ABB RAPID module: FML2H3SegmentOrg.mod

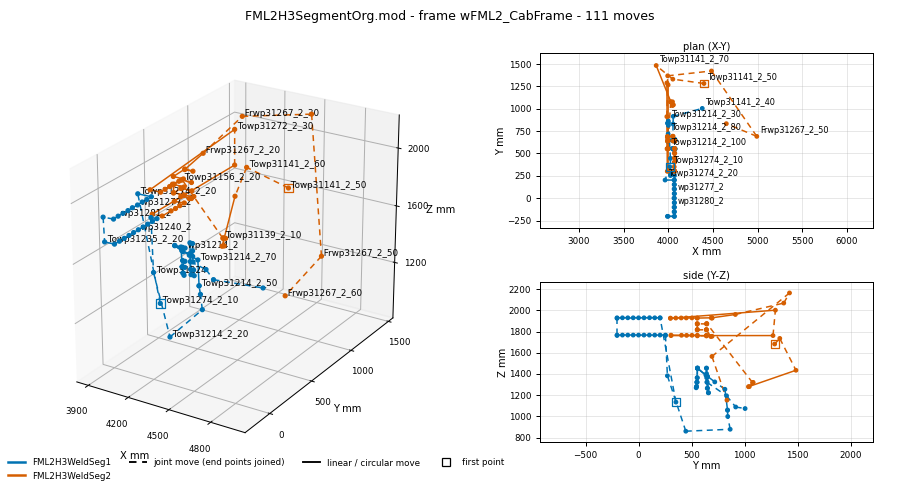
[picture p0: tool path of FML2H3SegmentOrg.mod in frame wFML2_CabFrame, 111 of 113 moves have a stored position in this frame; points joined in program order, loops and branches not executed]
%%%
   VERSION: 1
   LANGUAGE: ENGLISH
%%%

MODULE FML2H3Segment
  !
  !***********************************
  !*                                 *
  !*   Module : FML2H3Segment.mod    *
  !*   Name   : R2 2V6=V2=AR22       *
  !*   Task   : T_Rob1               *
  !*                                 *
  !***********************************
  !
  ! Rob 1 : irb 66-61388 \ 2V6=V2=AR22
  !
  !*********************
  ! Robtargets
  !*********************
  LOCAL CONST robtarget Towp31274_2_10:=[[4016.45,352.30,1134.15],[0.162794,-0.671420,0.154786,-0.706211],[0,-1,0,0],[9E9,100.000,9E9,9E9,9E9,9E9]];
  LOCAL CONST robtarget Towp31274_2_20:=[[3964.30,202.95,1926.71],[0.082443,-0.684548,0.078373,-0.720038],[-1,-1,0,0],[9E9,129.723,9E9,9E9,9E9,9E9]];
  LOCAL CONST robtarget wp31274_2:=[[4065.31,202.75,1929.60],[0.0644104,-0.686294,0.0612422,-0.721873],[-1,-1,0,0],[9E+09,25.0006,9E+09,9E+09,9E+09,9E+09]];
  LOCAL CONST robtarget Towp31275_2_10:=[[4050.21,151.97,1923.72],[0.064411,-0.686287,0.061241,-0.721867],[-1,-1,0,0],[9E9,30.000,9E9,9E9,9E9,9E9]];
  LOCAL CONST robtarget wp31275_2:=[[4065.68,152.48,1929.12],[0.0643992,-0.686292,0.0612485,-0.721875],[-1,-1,0,0],[9E+09,25.0001,9E+09,9E+09,9E+09,9E+09]];
  LOCAL CONST robtarget Towp31276_2_10:=[[4050.21,101.31,1923.72],[0.090401,-0.683647,0.085941,-0.719087],[-1,-1,0,0],[9E9,30.000,9E9,9E9,9E9,9E9]];
  LOCAL CONST robtarget wp31276_2:=[[4065.38,103.38,1930.02],[0.105651,-0.68166,0.100447,-0.716999],[-1,-1,0,0],[9E+09,25.001,9E+09,9E+09,9E+09,9E+09]];
  LOCAL CONST robtarget Towp31277_2_10:=[[4050.21,50.65,1923.72],[0.105651,-0.681667,0.100451,-0.717007],[-1,-1,0,0],[9E9,30.000,9E9,9E9,9E9,9E9]];
  LOCAL CONST robtarget wp31277_2:=[[4066.10,51.42,1929.09],[0.105652,-0.681659,0.100451,-0.717],[-1,-1,0,0],[9E+09,24.9997,9E+09,9E+09,9E+09,9E+09]];
  LOCAL CONST robtarget Towp31278_2_10:=[[4050.21,0.00,1923.72],[0.115181,-0.680257,0.109501,-0.715537],[-1,-1,0,0],[9E9,30.000,9E9,9E9,9E9,9E9]];
  LOCAL CONST robtarget wp31278_2:=[[4063.93,-0.02,1929.13],[0.115181,-0.680257,0.109501,-0.715537],[-1,-1,0,0],[9E9,25.000,9E9,9E9,9E9,9E9]];
  LOCAL CONST robtarget Towp31279_2_10:=[[4050.21,-50.65,1923.72],[0.131391,-0.677597,0.124921,-0.712737],[-1,-1,0,0],[9E9,30.000,9E9,9E9,9E9,9E9]];
  LOCAL CONST robtarget wp31279_2:=[[4066.40,-50.84,1929.14],[0.131392,-0.677596,0.124922,-0.712737],[-1,-1,0,0],[9E+09,25.0001,9E+09,9E+09,9E+09,9E+09]];
  LOCAL CONST robtarget Towp31280_2_10:=[[4050.21,-101.31,1923.72],[0.131391,-0.677597,0.124921,-0.712737],[-1,-1,0,0],[9E9,30.000,9E9,9E9,9E9,9E9]];
  LOCAL CONST robtarget wp31280_2:=[[4064.89,-101.49,1929.14],[0.131386,-0.677595,0.124923,-0.712739],[-1,-1,0,0],[9E+09,25.0001,9E+09,9E+09,9E+09,9E+09]];
  LOCAL CONST robtarget Towp31281_2_10:=[[4050.21,-151.97,1923.72],[0.144731,-0.675137,0.137601,-0.710147],[-1,-1,0,0],[9E9,30.000,9E9,9E9,9E9,9E9]];
  LOCAL CONST robtarget wp31281_2:=[[4065.09,-152.28,1929.13],[0.144727,-0.675136,0.137603,-0.710148],[-1,-1,0,0],[9E+09,25.0001,9E+09,9E+09,9E+09,9E+09]];
  LOCAL CONST robtarget Towp31282_2_10:=[[4050.21,-202.63,1923.72],[0.172142,-0.669297,0.163652,-0.704007],[-1,-1,0,0],[9E9,30.000,9E9,9E9,9E9,9E9]];
  LOCAL CONST robtarget wp31282_2:=[[4067.03,-203.17,1929.08],[0.16373,-0.671199,0.155666,-0.706012],[-1,-1,0,0],[9E+09,25.0001,9E+09,9E+09,9E+09,9E+09]];
  LOCAL CONST robtarget Towp31235_2_10:=[[3990.48,-202.94,1924.40],[0.146426,-0.674805,0.139211,-0.709801],[-1,-1,0,0],[9E9,100.000,9E9,9E9,9E9,9E9]];
  LOCAL CONST robtarget Towp31235_2_20:=[[3996.84,-202.94,1763.15],[0.141411,-0.692597,0.141321,-0.693067],[-1,-1,0,0],[9E9,100.000,9E9,9E9,9E9,9E9]];
  LOCAL CONST robtarget wp31235_2:=[[4069.18,-202.99,1765.78],[0.141408,-0.692595,0.141328,-0.693067],[-1,-1,0,0],[9E+09,25.0001,9E+09,9E+09,9E+09,9E+09]];
  LOCAL CONST robtarget Towp31236_2_10:=[[4054.42,-151.97,1759.49],[0.128101,-0.695197,0.128011,-0.695637],[-1,-1,0,0],[9E9,30.000,9E9,9E9,9E9,9E9]];
  LOCAL CONST robtarget wp31236_2:=[[4069.77,-152.16,1766.20],[0.128108,-0.695197,0.128004,-0.695632],[-1,-1,0,0],[9E+09,25.0001,9E+09,9E+09,9E+09,9E+09]];
  LOCAL CONST robtarget Towp31237_2_10:=[[4054.42,-101.31,1759.49],[0.128101,-0.695197,0.128011,-0.695637],[-1,-1,0,0],[9E9,30.000,9E9,9E9,9E9,9E9]];
  LOCAL CONST robtarget wp31237_2:=[[4070.38,-101.50,1766.20],[0.1281,-0.695194,0.128011,-0.695635],[-1,-1,0,0],[9E+09,24.9996,9E+09,9E+09,9E+09,9E+09]];
  LOCAL CONST robtarget Towp31238_2_10:=[[4054.41,-50.65,1759.49],[0.128381,-0.695127,0.128301,-0.695597],[-1,-1,0,0],[9E9,30.000,9E9,9E9,9E9,9E9]];
  LOCAL CONST robtarget wp31238_2:=[[4070.05,-50.84,1766.20],[0.128385,-0.695128,0.128301,-0.695595],[-1,-1,0,0],[9E+09,24.9986,9E+09,9E+09,9E+09,9E+09]];
  LOCAL CONST robtarget Towp31239_2_10:=[[4054.41,0.00,1759.49],[0.128101,-0.695197,0.128011,-0.695637],[-1,-1,0,0],[9E9,30.000,9E9,9E9,9E9,9E9]];
  LOCAL CONST robtarget wp31239_2:=[[4069.17,-0.19,1766.20],[0.128107,-0.695196,0.128006,-0.695633],[-1,-1,0,0],[9E+09,25.0001,9E+09,9E+09,9E+09,9E+09]];
  LOCAL CONST robtarget Towp31240_2_10:=[[4054.42,50.65,1759.49],[0.113601,-0.697707,0.113531,-0.698147],[-1,-1,0,0],[9E9,30.000,9E9,9E9,9E9,9E9]];
  LOCAL CONST robtarget wp31240_2:=[[4069.38,50.63,1766.22],[0.113599,-0.697707,0.113531,-0.698148],[-1,-1,0,0],[9E+09,24.9996,9E+09,9E+09,9E+09,9E+09]];
  LOCAL CONST robtarget Towp31241_2_10:=[[4054.42,101.31,1759.49],[0.113601,-0.697707,0.113531,-0.698147],[-1,-1,0,0],[9E9,30.000,9E9,9E9,9E9,9E9]];
  LOCAL CONST robtarget wp31241_2:=[[4070.30,101.27,1766.21],[0.113606,-0.697708,0.113529,-0.698146],[-1,-1,0,0],[9E+09,25.0001,9E+09,9E+09,9E+09,9E+09]];
  LOCAL CONST robtarget Towp31242_2_10:=[[4054.42,151.97,1759.49],[0.062941,-0.704077,0.062901,-0.704527],[-1,-1,0,0],[9E9,30.000,9E9,9E9,9E9,9E9]];
  LOCAL CONST robtarget wp31242_2:=[[4069.10,152.47,1766.17],[0.0629363,-0.704074,0.0629048,-0.704529],[-1,-1,0,0],[9E+09,25.0006,9E+09,9E+09,9E+09,9E+09]];
  LOCAL CONST robtarget Towp31243_2_10:=[[4054.42,202.62,1759.49],[0.113601,-0.697707,0.113531,-0.698147],[-1,-1,0,0],[9E9,30.000,9E9,9E9,9E9,9E9]];
  LOCAL CONST robtarget wp31243_2:=[[4069.64,202.57,1766.21],[0.113604,-0.697709,0.113531,-0.698146],[-1,-1,0,0],[9E+09,25.0006,9E+09,9E+09,9E+09,9E+09]];
  LOCAL CONST robtarget Towp31244_2_10:=[[4054.42,253.28,1759.49],[0.098771,-0.699977,0.098711,-0.700377],[-1,-1,0,0],[9E9,30.000,9E9,9E9,9E9,9E9]];
  LOCAL CONST robtarget wp31244_2:=[[4069.47,253.41,1766.22],[0.098779,-0.699981,0.0987012,-0.700377],[-1,-1,0,0],[9E+09,25.0001,9E+09,9E+09,9E+09,9E+09]];
  LOCAL CONST robtarget Towp31214_2_10:=[[4024.34,253.56,1763.19],[0.085541,-0.701915,0.085526,-0.701914],[-1,-1,0,0],[9E9,100.000,9E9,9E9,9E9,9E9]];
  LOCAL CONST robtarget Towp31214_2_20:=[[4024.15,445.26,859.90],[0.209663,-0.669229,0.163293,-0.693909],[0,-1,0,0],[9E9,30.000,9E9,9E9,9E9,9E9]];
  LOCAL CONST robtarget Towp31214_2_30:=[[4000.53,863.67,878.09],[0.209664,-0.669228,0.163288,-0.693910],[0,-1,1,0],[9E9,29.999,9E9,9E9,9E9,9E9]];
  LOCAL CONST robtarget Towp31214_2_40:=[[4001.68,840.75,998.57],[0.206529,-0.679094,0.209107,-0.672645],[0,-1,0,0],[9E9,74.423,9E9,9E9,9E9,9E9]];
  LOCAL CONST robtarget Towp31214_2_50:=[[3992.94,838.76,1058.72],[0.202837,-0.683610,0.236031,-0.660170],[0,-1,0,0],[9E9,99.999,9E9,9E9,9E9,9E9]];
  LOCAL CONST robtarget Towp31214_2_60:=[[3992.93,838.76,1058.72],[0.202842,-0.683617,0.236032,-0.660177],[0,-1,0,0],[9E9,100.000,9E9,9E9,9E9,9E9]];
  LOCAL CONST robtarget Towp31214_2_70:=[[4001.18,814.12,1255.53],[0.202842,-0.683617,0.236032,-0.660147],[0,-1,0,0],[9E9,100.000,9E9,9E9,9E9,9E9]];
  LOCAL CONST robtarget Towp31214_2_80:=[[3998.59,718.55,1324.71],[0.238582,-0.667717,0.261043,-0.655047],[-1,-1,0,0],[9E9,100.000,9E9,9E9,9E9,9E9]];
  LOCAL CONST robtarget Towp31214_2_90:=[[3996.43,634.65,1388.99],[0.301443,-0.639626,0.301443,-0.639626],[-1,0,-1,0],[9E9,100.000,9E9,9E9,9E9,9E9]];
  LOCAL CONST robtarget Towp31214_2_100:=[[3996.43,555.21,1454.56],[0.301443,-0.639626,0.301443,-0.639626],[-1,0,-1,0],[9E9,100.000,9E9,9E9,9E9,9E9]];
  LOCAL CONST robtarget wp31214_2:=[[4074.78,555.19,1454.58],[0.301448,-0.639635,0.301446,-0.63963],[-1,-1,0,0],[9E+09,25.0006,9E+09,9E+09,9E+09,9E+09]];
  LOCAL CONST robtarget Towp31216_2_10:=[[4055.43,555.21,1454.56],[0.301443,-0.639626,0.301443,-0.639626],[-1,0,-1,0],[9E9,30.000,9E9,9E9,9E9,9E9]];
  LOCAL CONST robtarget Towp31216_2_20:=[[4055.43,553.86,1363.93],[0.301443,-0.639626,0.301443,-0.639626],[-1,-1,0,0],[9E9,30.000,9E9,9E9,9E9,9E9]];
  LOCAL CONST robtarget wp31216_2:=[[4074.88,551.89,1363.92],[0.30144,-0.639615,0.301463,-0.639645],[-1,-1,0,0],[9E+09,25.0011,9E+09,9E+09,9E+09,9E+09]];
  LOCAL CONST robtarget Towp31217_2_10:=[[4053.93,550.53,1320.87],[0.301443,-0.639626,0.301443,-0.639626],[-1,-1,0,0],[9E9,30.000,9E9,9E9,9E9,9E9]];
  LOCAL CONST robtarget wp31217_2:=[[4074.70,550.51,1322.31],[0.301448,-0.639642,0.301439,-0.639626],[-1,-1,0,0],[9E+09,25.0006,9E+09,9E+09,9E+09,9E+09]];
  LOCAL CONST robtarget Towp31218_2_10:=[[4053.93,550.53,1320.87],[0.301443,-0.639626,0.301443,-0.639626],[-1,-1,0,0],[9E9,30.000,9E9,9E9,9E9,9E9]];
  LOCAL CONST robtarget Towp31218_2_20:=[[4066.88,546.50,1280.56],[0.414899,-0.572588,0.414893,-0.572595],[-1,0,-1,0],[9E9,29.999,9E9,9E9,9E9,9E9]];
  LOCAL CONST robtarget wp31218_2:=[[4072.69,543.03,1269.14],[0.414899,-0.572585,0.414894,-0.572598],[-1,0,-1,0],[9E+09,24.9991,9E+09,9E+09,9E+09,9E+09]];
  LOCAL CONST robtarget Towp31143_2_10:=[[4060.85,546.50,1280.50],[0.414897,-0.572601,0.414893,-0.572583],[-1,0,-1,0],[9E9,30.000,9E9,9E9,9E9,9E9]];
  LOCAL CONST robtarget Towp31143_2_20:=[[4043.07,555.22,1454.48],[0.301450,-0.639637,0.301445,-0.639627],[-1,-1,0,0],[9E9,56.519,9E9,9E9,9E9,9E9]];
  LOCAL CONST robtarget Towp31143_2_30:=[[3996.29,555.12,1452.38],[0.302913,-0.638946,0.302913,-0.638946],[-1,0,-1,0],[9E9,100.000,9E9,9E9,9E9,9E9]];
  LOCAL CONST robtarget Towp31143_2_40:=[[3996.29,649.96,1374.83],[0.302913,-0.638946,0.302913,-0.638946],[-1,0,-1,0],[9E9,100.000,9E9,9E9,9E9,9E9]];
  LOCAL CONST robtarget Towp31143_2_50:=[[4049.79,649.96,1374.83],[0.302913,-0.638946,0.302913,-0.638946],[-1,0,-1,0],[9E9,100.000,9E9,9E9,9E9,9E9]];
  LOCAL CONST robtarget Towp31143_2_60:=[[4048.93,659.76,1222.18],[0.404844,-0.579746,0.404844,-0.579746],[-1,0,-1,0],[9E9,30.000,9E9,9E9,9E9,9E9]];
  LOCAL CONST robtarget wp31143_2:=[[4074.64,657.65,1222.13],[0.404851,-0.579739,0.404851,-0.579737],[-1,0,-1,0],[9E+09,25.0006,9E+09,9E+09,9E+09,9E+09]];
  LOCAL CONST robtarget Towp31144_2_10:=[[4055.00,650.35,1263.04],[0.404844,-0.579746,0.404844,-0.579746],[-1,0,-1,0],[9E9,30.000,9E9,9E9,9E9,9E9]];
  LOCAL CONST robtarget wp31144_2:=[[4075.34,650.28,1265.40],[0.404844,-0.579734,0.40484,-0.579754],[-1,0,-1,0],[9E+09,25.0006,9E+09,9E+09,9E+09,9E+09]];
  LOCAL CONST robtarget Towp31148_2_10:=[[4053.93,647.44,1265.33],[0.404844,-0.579746,0.404844,-0.579746],[-1,0,-1,0],[9E9,30.000,9E9,9E9,9E9,9E9]];
  LOCAL CONST robtarget Towp31148_2_20:=[[4055.43,640.80,1454.56],[0.301443,-0.639626,0.301443,-0.639626],[-1,0,-1,0],[9E9,30.000,9E9,9E9,9E9,9E9]];
  LOCAL CONST robtarget wp31148_2:=[[4075.85,639.45,1454.59],[0.30144,-0.639621,0.301448,-0.639647],[-1,0,-1,0],[9E+09,24.9996,9E+09,9E+09,9E+09,9E+09]];
  LOCAL CONST robtarget Towp31147_2_10:=[[4056.50,644.08,1399.66],[0.301443,-0.639626,0.301443,-0.639626],[-1,0,-1,0],[9E9,30.000,9E9,9E9,9E9,9E9]];
  LOCAL CONST robtarget wp31147_2:=[[4075.11,640.62,1402.76],[0.301453,-0.639626,0.301456,-0.639632],[-1,-1,0,0],[9E+09,25.0011,9E+09,9E+09,9E+09,9E+09]];
  LOCAL CONST robtarget Towp31146_2_10:=[[4056.50,644.14,1360.80],[0.301443,-0.639626,0.301443,-0.639626],[-1,0,-1,0],[9E9,30.000,9E9,9E9,9E9,9E9]];
  LOCAL CONST robtarget wp31146_2:=[[4074.31,642.12,1363.96],[0.301442,-0.639624,0.30145,-0.639641],[-1,-1,0,0],[9E+09,25.0006,9E+09,9E+09,9E+09,9E+09]];
  LOCAL CONST robtarget Towp31145_2_10:=[[4055.00,647.57,1317.86],[0.329033,-0.625896,0.329033,-0.625896],[-1,0,-1,0],[9E9,30.000,9E9,9E9,9E9,9E9]];
  LOCAL CONST robtarget wp31145_2:=[[4075.02,645.18,1323.40],[0.329045,-0.625872,0.329049,-0.625892],[-1,0,-1,0],[9E+09,25.0001,9E+09,9E+09,9E+09,9E+09]];
  LOCAL CONST robtarget Towp31141_2_10:=[[4053.93,645.31,1320.69],[0.329033,-0.625896,0.329033,-0.625896],[-1,0,-1,0],[9E9,30.000,9E9,9E9,9E9,9E9]];
  LOCAL CONST robtarget Towp31141_2_20:=[[4053.93,829.43,1193.98],[0.329033,-0.625896,0.329033,-0.625896],[-1,0,-1,0],[9E9,50.000,9E9,9E9,9E9,9E9]];
  LOCAL CONST robtarget Towp31141_2_30:=[[4055.61,915.71,1088.15],[0.311158,-0.574108,0.357827,-0.667488],[-1,0,-1,0],[9E9,49.997,9E9,9E9,9E9,9E9]];
  LOCAL CONST robtarget Towp31141_2_40:=[[4380.43,1004.47,1073.50],[0.329033,-0.625896,0.329033,-0.625896],[-1,0,-1,0],[9E9,50.000,9E9,9E9,9E9,9E9]];
  LOCAL CONST robtarget Towp31141_2_50:=[[4399.60,1283.05,1681.87],[0.242317,-0.631638,0.388427,-0.625652],[-2,0,-1,0],[9E9,48.091,9E9,9E9,9E9,9E9]];
  LOCAL CONST robtarget Towp31141_2_60:=[[4051.14,1331.48,1734.78],[0.322441,-0.595529,0.421583,-0.603029],[-2,0,-1,0],[9E9,48.372,9E9,9E9,9E9,9E9]];
  LOCAL CONST robtarget Towp31141_2_70:=[[3865.02,1484.04,1434.51],[0.607774,-0.566534,0.442110,-0.337919],[-2,0,-2,0],[9E9,66.407,9E9,9E9,9E9,9E9]];
  LOCAL CONST robtarget Towp31141_2_80:=[[4046.26,1036.05,1279.43],[0.624891,-0.566993,0.438571,-0.309331],[-2,0,-2,0],[9E9,105.850,9E9,9E9,9E9,9E9]];
  LOCAL CONST robtarget wp31141_2:=[[4057.63,1044.03,1280.67],[0.624912,-0.586047,0.421153,-0.297766],[-2,0,-2,0],[9E+09,25.0006,9E+09,9E+09,9E+09,9E+09]];
  LOCAL CONST robtarget Towp31139_2_10:=[[4028.65,1078.45,1319.83],[0.493609,-0.505141,0.494963,-0.506156],[-2,0,-2,0],[9E+09,40,9E+09,9E+09,9E+09,9E+09]];
  LOCAL CONST robtarget wp31139_2:=[[4047.28,1078.46,1319.97],[0.493612,-0.505140,0.494959,-0.506158],[-2,0,-2,0],[9E9,25.000,9E9,9E9,9E9,9E9]];
  LOCAL CONST robtarget Towp31156_2_10:=[[4027.10,1076.22,1316.29],[0.496076,-0.505810,0.494748,-0.503278],[-2,0,-2,0],[9E9,82.552,9E9,9E9,9E9,9E9]];
  LOCAL CONST robtarget Towp31156_2_20:=[[3999.20,643.27,1874.83],[0.41306,-0.570139,0.400218,-0.586642],[-1,0,-1,0],[9E+09,128.149,9E+09,9E+09,9E+09,9E+09]];
  LOCAL CONST robtarget wp31156_2:=[[4071.98,640.13,1872.87],[0.413058,-0.570143,0.400228,-0.586633],[-1,0,-1,0],[9E+09,24.998,9E+09,9E+09,9E+09,9E+09]];
  LOCAL CONST robtarget Towp31206_2_10:=[[3993.72,643.17,1870.74],[0.413056,-0.570144,0.40022,-0.586639],[-1,0,-1,0],[9E+09,100.002,9E+09,9E+09,9E+09,9E+09]];
  LOCAL CONST robtarget Towp31206_2_20:=[[3986.60,552.91,1873.31],[0.420259,-0.563937,0.407544,-0.582465],[-1,0,-1,0],[9E+09,100.001,9E+09,9E+09,9E+09,9E+09]];
  LOCAL CONST robtarget wp31206_2:=[[4072.95,553.58,1873.34],[0.420258,-0.563936,0.40753,-0.582476],[-1,0,-1,0],[9E+09,25.1416,9E+09,9E+09,9E+09,9E+09]];
  LOCAL CONST robtarget Towp31207_2_10:=[[3992.65,553.82,1869.80],[0.420261,-0.563933,0.407546,-0.582466],[-1,0,-1,0],[9E9,100.000,9E9,9E9,9E9,9E9]];
  LOCAL CONST robtarget Towp31207_2_20:=[[3993.78,553.55,1816.78],[0.448931,-0.544821,0.443606,-0.552127],[-1,0,-1,0],[9E+09,100.001,9E+09,9E+09,9E+09,9E+09]];
  LOCAL CONST robtarget wp31207_2:=[[4071.90,554.05,1818.23],[0.448933,-0.544814,0.443612,-0.552128],[-1,0,-1,0],[9E+09,25.0015,9E+09,9E+09,9E+09,9E+09]];
  LOCAL CONST robtarget Towp31155_2_10:=[[3993.78,552.83,1815.08],[0.448933,-0.544818,0.443605,-0.55213],[-1,0,-1,0],[9E+09,99.9996,9E+09,9E+09,9E+09,9E+09]];
  LOCAL CONST robtarget Towp31155_2_20:=[[3993.77,638.71,1816.62],[0.431159,-0.559379,0.425412,-0.56588],[-1,0,-1,0],[9E+09,100.001,9E+09,9E+09,9E+09,9E+09]];
  LOCAL CONST robtarget wp31155_2:=[[4074.77,639.89,1817.01],[0.431155,-0.559381,0.425402,-0.56589],[-1,0,-1,0],[9E+09,24.9996,9E+09,9E+09,9E+09,9E+09]];
  LOCAL CONST robtarget Towp31250_2_10:=[[3993.76,638.70,1816.62],[0.431161,-0.559377,0.425412,-0.565881],[-1,0,-1,0],[9E+09,100.001,9E+09,9E+09,9E+09,9E+09]];
  LOCAL CONST robtarget Towp31250_2_20:=[[3989.70,680.85,1752.63],[0.515328,-0.560652,0.415979,-0.497059],[-2,0,-2,0],[9E9,100.000,9E9,9E9,9E9,9E9]];
  LOCAL CONST robtarget wp31250_2:=[[4054.17,692.94,1754.95],[0.499526,-0.571079,0.416555,-0.500823],[-2,0,-2,0],[9E+09,4.63808,9E+09,9E+09,9E+09,9E+09]];
  LOCAL CONST robtarget Towp31154_10:=[[4054.88,639.53,1759.33],[0.449086,-0.544740,0.445578,-0.550491],[-1,0,-1,0],[9E9,30.000,9E9,9E9,9E9,9E9]];
  LOCAL CONST robtarget wp31154:=[[4071.23,639.50,1763.81],[0.446935,-0.546472,0.443467,-0.552227],[-1,0,-1,0],[9E+09,25.0011,9E+09,9E+09,9E+09,9E+09]];
  LOCAL CONST robtarget Towp31208_2_10:=[[3990.99,639.69,1758.85],[0.440179,-0.551840,0.436783,-0.557616],[-1,0,-1,0],[9E9,100.000,9E9,9E9,9E9,9E9]];
  LOCAL CONST robtarget Towp31208_2_20:=[[3998.00,554.01,1758.87],[0.436139,-0.555460,0.431739,-0.561113],[-1,0,-1,0],[9E9,100.000,9E9,9E9,9E9,9E9]];
  LOCAL CONST robtarget wp31208_2:=[[4073.29,554.09,1764.50],[0.418898,-0.568302,0.414662,-0.574119],[-1,0,-1,0],[9E+09,24.9991,9E+09,9E+09,9E+09,9E+09]];
  LOCAL CONST robtarget Towp31249_2_10:=[[4054.40,506.52,1759.39],[0.420905,-0.568114,0.420622,-0.568473],[-1,0,-1,0],[9E9,30.000,9E9,9E9,9E9,9E9]];
  LOCAL CONST robtarget wp31249_2:=[[4073.14,503.35,1764.12],[0.445274,-0.549243,0.444983,-0.549594],[-1,0,-1,0],[9E+09,25.0011,9E+09,9E+09,9E+09,9E+09]];
  LOCAL CONST robtarget Towp31248_2_10:=[[4054.35,455.87,1759.37],[0.442975,-0.551095,0.442670,-0.551462],[-1,0,-1,0],[9E9,30.000,9E9,9E9,9E9,9E9]];
  LOCAL CONST robtarget wp31248_2:=[[4074.33,452.68,1763.43],[0.443095,-0.550993,0.4428,-0.551364],[-1,0,-1,0],[9E+09,25.0006,9E+09,9E+09,9E+09,9E+09]];
  LOCAL CONST robtarget Towp31247_2_10:=[[4054.43,405.23,1759.44],[0.433900,-0.558272,0.433608,-0.558612],[-1,0,-1,0],[9E9,30.000,9E9,9E9,9E9,9E9]];
  LOCAL CONST robtarget wp31247_2:=[[4072.88,404.67,1764.30],[0.44457,-0.549815,0.444266,-0.550171],[-1,0,-1,0],[9E+09,25.0006,9E+09,9E+09,9E+09,9E+09]];
  LOCAL CONST robtarget Towp31245_2_10:=[[4054.33,308.91,1759.42],[0.445533,-0.549029,0.445229,-0.549398],[-1,0,-1,0],[9E9,30.000,9E9,9E9,9E9,9E9]];
  LOCAL CONST robtarget wp31245_2:=[[4073.04,305.67,1765.58],[0.442311,-0.551633,0.442006,-0.55199],[-1,0,-1,0],[9E+09,25.0011,9E+09,9E+09,9E+09,9E+09]];
  LOCAL CONST robtarget Towp31272_2_10:=[[3998.39,305.75,1761.34],[0.443862,-0.550393,0.443569,-0.550727],[-1,0,-1,0],[9E9,100.000,9E9,9E9,9E9,9E9]];
  LOCAL CONST robtarget Towp31272_2_20:=[[3998.33,1267.50,1761.67],[0.408729,-0.576926,0.408449,-0.577292],[-2,0,-2,0],[9E9,100.000,9E9,9E9,9E9,9E9]];
  LOCAL CONST robtarget Towp31272_2_30:=[[3984.69,1290.11,2001.11],[0.485005,-0.510893,0.428801,-0.565586],[-2,0,-2,0],[9E9,99.999,9E9,9E9,9E9,9E9]];
  LOCAL CONST robtarget Towp31272_2_40:=[[3989.09,300.38,1924.69],[0.521335,-0.478625,0.495645,-0.503455],[-1,0,-1,0],[9E9,100.000,9E9,9E9,9E9,9E9]];
  LOCAL CONST robtarget wp31272_2:=[[4067.79,300.37,1925.97],[0.521332,-0.478634,0.495635,-0.503456],[-1,0,-1,0],[9E+09,25.0001,9E+09,9E+09,9E+09,9E+09]];
  LOCAL CONST robtarget Towp31271_2_10:=[[4050.21,354.61,1923.72],[0.521335,-0.478645,0.495645,-0.503455],[-1,0,-1,0],[9E9,30.000,9E9,9E9,9E9,9E9]];
  LOCAL CONST robtarget wp31271_2:=[[4066.84,351.01,1926.91],[0.521334,-0.478636,0.495637,-0.503451],[-1,0,-1,0],[9E+09,25.0001,9E+09,9E+09,9E+09,9E+09]];
  LOCAL CONST robtarget Towp31270_2_10:=[[4050.21,405.27,1923.72],[0.521335,-0.478645,0.495645,-0.503455],[-1,0,-1,0],[9E9,30.000,9E9,9E9,9E9,9E9]];
  LOCAL CONST robtarget wp31270_2:=[[4066.97,401.71,1927.73],[0.521328,-0.478638,0.495633,-0.503458],[-1,0,-1,0],[9E+09,25.0001,9E+09,9E+09,9E+09,9E+09]];
  LOCAL CONST robtarget Towp31269_2_10:=[[4050.21,455.93,1923.72],[0.521335,-0.478645,0.495645,-0.503455],[-1,0,-1,0],[9E9,30.000,9E9,9E9,9E9,9E9]];
  LOCAL CONST robtarget wp31269_2:=[[4068.97,449.38,1927.88],[0.521329,-0.478638,0.495635,-0.503456],[-1,0,-1,0],[9E+09,25.0001,9E+09,9E+09,9E+09,9E+09]];
  LOCAL CONST robtarget Towp31268_2_10:=[[4050.21,506.59,1923.72],[0.521335,-0.478645,0.495645,-0.503455],[-1,0,-1,0],[9E9,30.000,9E9,9E9,9E9,9E9]];
  LOCAL CONST robtarget wp31268_2:=[[4068.26,502.99,1928.11],[0.521335,-0.478633,0.495632,-0.503457],[-1,0,-1,0],[9E+09,25.0006,9E+09,9E+09,9E+09,9E+09]];
  LOCAL CONST robtarget Towp31205_2_10:=[[4051.57,557.20,1924.47],[0.517945,-0.481745,0.487075,-0.512265],[-1,0,-1,0],[9E9,30.000,9E9,9E9,9E9,9E9]];
  LOCAL CONST robtarget wp31205_2:=[[4069.45,552.93,1926.78],[0.517952,-0.48173,0.487074,-0.51227],[-1,0,-1,0],[9E+09,25.0011,9E+09,9E+09,9E+09,9E+09]];
  LOCAL CONST robtarget Towp31267_2_10:=[[3993.41,553.66,1926.43],[0.517945,-0.481745,0.487075,-0.512265],[-1,0,-1,0],[9E9,100.000,9E9,9E9,9E9,9E9]];
  LOCAL CONST robtarget Towp31267_2_20:=[[3990.15,691.03,1929.16],[0.571776,-0.495345,0.491885,-0.430994],[-2,0,-2,0],[9E9,100.000,9E9,9E9,9E9,9E9]];
  LOCAL CONST robtarget wp31267_2:=[[4048.88,693.20,1926.26],[0.571776,-0.495344,0.491883,-0.430997],[-2,0,-2,0],[9E9,24.999,9E9,9E9,9E9,9E9]];
  LOCAL CONST robtarget Frwp31267_2_10:=[[3992.59,685.11,1928.11],[0.571776,-0.495345,0.491885,-0.430994],[-2,0,-2,0],[9E9,100.000,9E9,9E9,9E9,9E9]];
  LOCAL CONST robtarget Frwp31267_2_20:=[[3984.19,912.55,1960.54],[0.515098,-0.552535,0.426442,-0.497521],[-2,0,-2,0],[9E9,100.001,9E9,9E9,9E9,9E9]];
  LOCAL CONST robtarget Frwp31267_2_30:=[[3993.68,1368.95,2068.12],[0.440251,-0.613027,0.356615,-0.550638],[-2,0,-2,0],[9E9,100.000,9E9,9E9,9E9,9E9]];
  LOCAL CONST robtarget Frwp31267_2_40:=[[4483.73,1423.17,2163.62],[0.282020,-0.710709,0.244498,-0.596303],[-2,0,-1,0],[9E9,99.999,9E9,9E9,9E9,9E9]];
  LOCAL CONST robtarget Frwp31267_2_50:=[[4990.52,691.63,1564.75],[0.303425,-0.707680,0.184932,-0.610674],[-1,-1,0,0],[9E9,29.997,9E9,9E9,9E9,9E9]];
  LOCAL CONST robtarget Frwp31267_2_60:=[[4649.39,833.49,1152.96],[0.385471,-0.603349,-0.013916,-0.697989],[0,-1,0,0],[9E9,58.131,9E9,9E9,9E9,9E9]];
  !
  !*********************
  ! SpotData
  !*********************
  LOCAL PERS spotdata Sd_wp31274_2_20:=[3127422,0,0,0,0];
  LOCAL PERS spotdata Sd_wp31275_2_20:=[3127522,0,0,0,0];
  LOCAL PERS spotdata Sd_wp31276_2_20:=[3127622,0,0,0,0];
  LOCAL PERS spotdata Sd_wp31277_2_20:=[3127722,0,0,0,0];
  LOCAL PERS spotdata Sd_wp31278_2_20:=[3127822,0,0,0,0];
  LOCAL PERS spotdata Sd_wp31279_2_20:=[3127922,0,0,0,0];
  LOCAL PERS spotdata Sd_wp31280_2_20:=[3128022,0,0,0,0];
  LOCAL PERS spotdata Sd_wp31281_2_20:=[3128122,0,0,0,0];
  LOCAL PERS spotdata Sd_wp31282_2_20:=[3128222,0,0,0,0];
  LOCAL PERS spotdata Sd_wp31235_2_20:=[3123522,0,0,0,0];
  LOCAL PERS spotdata Sd_wp31236_2_20:=[3123622,0,0,0,0];
  LOCAL PERS spotdata Sd_wp31237_2_20:=[3123722,0,0,0,0];
  LOCAL PERS spotdata Sd_wp31238_2_20:=[3123822,0,0,0,0];
  LOCAL PERS spotdata Sd_wp31239_2_20:=[3123922,0,0,0,0];
  LOCAL PERS spotdata Sd_wp31240_2_20:=[3124022,0,0,0,0];
  LOCAL PERS spotdata Sd_wp31241_2_20:=[3124122,0,0,0,0];
  LOCAL PERS spotdata Sd_wp31242_2_20:=[3124222,0,0,0,0];
  LOCAL PERS spotdata Sd_wp31243_2_20:=[3124322,0,0,0,0];
  LOCAL PERS spotdata Sd_wp31244_2_20:=[3124422,0,0,0,0];
  LOCAL PERS spotdata Sd_wp31214_2_20:=[3121422,0,0,0,0];
  LOCAL PERS spotdata Sd_wp31216_2_20:=[3121622,0,0,0,0];
  LOCAL PERS spotdata Sd_wp31217_2_20:=[3121722,0,0,0,0];
  LOCAL PERS spotdata Sd_wp31218_2_20:=[3121822,0,0,0,0];
  LOCAL PERS spotdata Sd_wp31143_2_20:=[3114322,0,0,0,0];
  LOCAL PERS spotdata Sd_wp31144_2_20:=[3114422,0,0,0,0];
  LOCAL PERS spotdata Sd_wp31148_2_20:=[3114822,0,0,0,0];
  LOCAL PERS spotdata Sd_wp31147_2_20:=[3114722,0,0,0,0];
  LOCAL PERS spotdata Sd_wp31146_2_20:=[3114622,0,0,0,0];
  LOCAL PERS spotdata Sd_wp31145_2_20:=[3114522,0,0,0,0];
  LOCAL PERS spotdata Sd_wp31141_2_20:=[3114122,0,0,0,0];
  LOCAL PERS spotdata Sd_wp31139_2_20:=[3113922,0,0,0,0];
  LOCAL PERS spotdata Sd_wp31156_2_20:=[3115622,0,0,0,0];
  LOCAL PERS spotdata Sd_wp31206_2_20:=[3120622,0,0,0,0];
  LOCAL PERS spotdata Sd_wp31207_2_20:=[3120722,0,0,0,0];
  LOCAL PERS spotdata Sd_wp31155_2_20:=[3115522,0,0,0,0];
  LOCAL PERS spotdata Sd_wp31250_2_20:=[3125022,0,0,0,0];
  LOCAL PERS spotdata Sd_wp31154_20:=[3115420,0,0,0,0];
  LOCAL PERS spotdata Sd_wp31208_2_20:=[3120822,0,0,0,0];
  LOCAL PERS spotdata Sd_wp31249_2_20:=[3124922,0,0,0,0];
  LOCAL PERS spotdata Sd_wp31248_2_20:=[3124822,0,0,0,0];
  LOCAL PERS spotdata Sd_wp31247_2_20:=[3124722,0,0,0,0];
  LOCAL PERS spotdata Sd_wp31245_2_20:=[3124522,0,0,0,0];
  LOCAL PERS spotdata Sd_wp31272_2_20:=[3127222,0,0,0,0];
  LOCAL PERS spotdata Sd_wp31271_2_20:=[3127122,0,0,0,0];
  LOCAL PERS spotdata Sd_wp31270_2_20:=[3127022,0,0,0,0];
  LOCAL PERS spotdata Sd_wp31269_2_20:=[3126922,0,0,0,0];
  LOCAL PERS spotdata Sd_wp31268_2_20:=[3126822,0,0,0,0];
  LOCAL PERS spotdata Sd_wp31205_2_20:=[3120522,0,0,0,0];
  LOCAL PERS spotdata Sd_wp31267_2_20:=[3126722,0,0,0,0];
  !!
  !
  !
  CONST robtarget Towp31224:=[[4024.01,271.77,1382.50],[0.137298,-0.691858,0.119416,-0.698728],[0,-1,0,0],[9E9,75.073,9E9,9E9,9E9,9E9]];
  !
  !----------------
  ! Part : FM L2 H3 - PHL
  !----------------
PROC FML2H3WeldSeg1()
    MoveAbsJ HomeXQ11Gun,vmax,fine,XQ11GunTCP\WObj:=wFML2_CabFrame;
    MoveJ Towp31274_2_10, v500, z30, XQ11GunTCP\WObj:=wFML2_CabFrame;
    MoveJ Towp31274_2_20, v500, z30, XQ11GunTCP\WObj:=wFML2_CabFrame;
    SpotL wp31274_2,vmax,XQ11Gun,Sd_wp31274_2_20\QuickRelease,XQ11GunTCP\WObj:=wFML2_CabFrame;
    SpotL wp31275_2,vmax,XQ11Gun,Sd_wp31275_2_20\QuickRelease,XQ11GunTCP\WObj:=wFML2_CabFrame;
    SpotL wp31276_2,vmax,XQ11Gun,Sd_wp31276_2_20\QuickRelease,XQ11GunTCP\WObj:=wFML2_CabFrame;
    SpotL wp31277_2,vmax,XQ11Gun,Sd_wp31277_2_20\QuickRelease,XQ11GunTCP\WObj:=wFML2_CabFrame;
    SpotL wp31278_2,vmax,XQ11Gun,Sd_wp31278_2_20\QuickRelease,XQ11GunTCP\WObj:=wFML2_CabFrame;
    SpotL wp31279_2,vmax,XQ11Gun,Sd_wp31279_2_20\QuickRelease,XQ11GunTCP\WObj:=wFML2_CabFrame;
    SpotL wp31280_2,vmax,XQ11Gun,Sd_wp31280_2_20\QuickRelease,XQ11GunTCP\WObj:=wFML2_CabFrame;
    SpotL wp31281_2,vmax,XQ11Gun,Sd_wp31281_2_20\QuickRelease,XQ11GunTCP\WObj:=wFML2_CabFrame;
    SpotL wp31282_2,vmax,XQ11Gun,Sd_wp31282_2_20\QuickRelease,XQ11GunTCP\WObj:=wFML2_CabFrame;
    MoveJ Towp31235_2_10,vmax,z30,XQ11GunTCP\WObj:=wFML2_CabFrame;
    MoveJ Towp31235_2_20,vmax,z30,XQ11GunTCP\WObj:=wFML2_CabFrame;
    SpotL wp31235_2,vmax,XQ11Gun,Sd_wp31235_2_20\QuickRelease,XQ11GunTCP\WObj:=wFML2_CabFrame;
    SpotL wp31236_2,vmax,XQ11Gun,Sd_wp31236_2_20\QuickRelease,XQ11GunTCP\WObj:=wFML2_CabFrame;
    SpotL wp31237_2,vmax,XQ11Gun,Sd_wp31237_2_20\QuickRelease,XQ11GunTCP\WObj:=wFML2_CabFrame;
    SpotL wp31238_2,vmax,XQ11Gun,Sd_wp31238_2_20\QuickRelease,XQ11GunTCP\WObj:=wFML2_CabFrame;
    SpotL wp31239_2,vmax,XQ11Gun,Sd_wp31239_2_20\QuickRelease,XQ11GunTCP\WObj:=wFML2_CabFrame;
    SpotL wp31240_2,vmax,XQ11Gun,Sd_wp31240_2_20\QuickRelease,XQ11GunTCP\WObj:=wFML2_CabFrame;
    SpotL wp31241_2,vmax,XQ11Gun,Sd_wp31241_2_20\QuickRelease,XQ11GunTCP\WObj:=wFML2_CabFrame;
    SpotL wp31242_2,vmax,XQ11Gun,Sd_wp31242_2_20\QuickRelease,XQ11GunTCP\WObj:=wFML2_CabFrame;
    SpotL wp31243_2,vmax,XQ11Gun,Sd_wp31243_2_20\QuickRelease,XQ11GunTCP\WObj:=wFML2_CabFrame;
    SpotL wp31244_2,vmax,XQ11Gun,Sd_wp31244_2_20\QuickRelease,XQ11GunTCP\WObj:=wFML2_CabFrame;
    MoveJ Towp31214_2_10,vmax,z30,XQ11GunTCP\WObj:=wFML2_CabFrame;
    MoveJ Towp31224, vmax, z30, XQ11GunTCP\WObj:=wFML2_CabFrame;
    MoveJ Towp31214_2_20,vmax,z30,XQ11GunTCP\WObj:=wFML2_CabFrame;
    MoveJ Towp31214_2_30,vmax,z30,XQ11GunTCP\WObj:=wFML2_CabFrame;
    MoveJ Towp31214_2_40,vmax,z30,XQ11GunTCP\WObj:=wFML2_CabFrame;
    MoveJ Towp31214_2_50,vmax,z30,XQ11GunTCP\WObj:=wFML2_CabFrame;
    MoveJ Towp31214_2_60,vmax,z30,XQ11GunTCP\WObj:=wFML2_CabFrame;
    MoveL Towp31214_2_70,vmax,z30,XQ11GunTCP\WObj:=wFML2_CabFrame;
    MoveJ Towp31214_2_80,vmax,z30,XQ11GunTCP\WObj:=wFML2_CabFrame;
    MoveL Towp31214_2_90,vmax,z30,XQ11GunTCP\WObj:=wFML2_CabFrame;
    MoveL Towp31214_2_100,vmax,z30,XQ11GunTCP\WObj:=wFML2_CabFrame;
    SpotL wp31214_2,vmax,XQ11Gun,Sd_wp31214_2_20\QuickRelease,XQ11GunTCP\WObj:=wFML2_CabFrame;
    MoveJ Towp31216_2_10,vmax,z30,XQ11GunTCP\WObj:=wFML2_CabFrame;
    MoveJ Towp31216_2_20,vmax,z30,XQ11GunTCP\WObj:=wFML2_CabFrame;
    SpotL wp31216_2,vmax,XQ11Gun,Sd_wp31216_2_20\QuickRelease,XQ11GunTCP\WObj:=wFML2_CabFrame;
    MoveJ Towp31217_2_10,vmax,z30,XQ11GunTCP\WObj:=wFML2_CabFrame;
    SpotL wp31217_2,vmax,XQ11Gun,Sd_wp31217_2_20\QuickRelease,XQ11GunTCP\WObj:=wFML2_CabFrame;
    MoveJ Towp31218_2_10,vmax,z30,XQ11GunTCP\WObj:=wFML2_CabFrame;
    MoveL Towp31218_2_20,vmax,z30,XQ11GunTCP\WObj:=wFML2_CabFrame;
    SpotL wp31218_2,vmax,XQ11Gun,Sd_wp31218_2_20\QuickRelease,XQ11GunTCP\WObj:=wFML2_CabFrame;
    MoveL Towp31143_2_10,vmax,z30,XQ11GunTCP\WObj:=wFML2_CabFrame;
    MoveL Towp31143_2_20,vmax,z30,XQ11GunTCP\WObj:=wFML2_CabFrame;
    MoveJ Towp31143_2_30,vmax,z30,XQ11GunTCP\WObj:=wFML2_CabFrame;
    MoveL Towp31143_2_40,vmax,z30,XQ11GunTCP\WObj:=wFML2_CabFrame;
    MoveJ Towp31143_2_50,vmax,z30,XQ11GunTCP\WObj:=wFML2_CabFrame;
    MoveL Towp31143_2_60,vmax,z30,XQ11GunTCP\WObj:=wFML2_CabFrame;
    SpotL wp31143_2,vmax,XQ11Gun,Sd_wp31143_2_20\QuickRelease,XQ11GunTCP\WObj:=wFML2_CabFrame;
    SpotL wp31144_2,vmax,XQ11Gun,Sd_wp31144_2_20\QuickRelease,XQ11GunTCP\WObj:=wFML2_CabFrame;
    MoveJ Towp31148_2_10,vmax,z30,XQ11GunTCP\WObj:=wFML2_CabFrame;
    MoveL Towp31148_2_20,vmax,z30,XQ11GunTCP\WObj:=wFML2_CabFrame;
    SpotL wp31148_2,vmax,XQ11Gun,Sd_wp31148_2_20\QuickRelease,XQ11GunTCP\WObj:=wFML2_CabFrame;
    SpotL wp31147_2,vmax,XQ11Gun,Sd_wp31147_2_20\QuickRelease,XQ11GunTCP\WObj:=wFML2_CabFrame;
    SpotL wp31146_2,vmax,XQ11Gun,Sd_wp31146_2_20\QuickRelease,XQ11GunTCP\WObj:=wFML2_CabFrame;
    SpotL wp31145_2,vmax,XQ11Gun,Sd_wp31145_2_20\QuickRelease,XQ11GunTCP\WObj:=wFML2_CabFrame;
    MoveJ Towp31141_2_10,vmax,z30,XQ11GunTCP\WObj:=wFML2_CabFrame;
    MoveJ Towp31141_2_20,vmax,z30,XQ11GunTCP\WObj:=wFML2_CabFrame;
    MoveJ Towp31141_2_30,vmax,z30,XQ11GunTCP\WObj:=wFML2_CabFrame;
    MoveJ Towp31141_2_40,vmax,z30,XQ11GunTCP\WObj:=wFML2_CabFrame;
ENDPROC
PROC FML2H3WeldSeg2()
    MoveJ Towp31141_2_50,vmax,z30,XQ11GunTCP\WObj:=wFML2_CabFrame;
    MoveJ Towp31141_2_60,vmax,z30,XQ11GunTCP\WObj:=wFML2_CabFrame;
    MoveJ Towp31141_2_70,vmax,z30,XQ11GunTCP\WObj:=wFML2_CabFrame;
    MoveL Towp31141_2_80,vmax,z30,XQ11GunTCP\WObj:=wFML2_CabFrame;
    SpotL wp31141_2, vmax, XQ11Gun, Sd_wp31141_2_20, XQ11GunTCP\WObj:=wFML2_CabFrame;
    MoveL Towp31139_2_10,vmax,z30,XQ11GunTCP\WObj:=wFML2_CabFrame;
    SpotL wp31139_2,vmax,XQ11Gun,Sd_wp31139_2_20\QuickRelease,XQ11GunTCP\WObj:=wFML2_CabFrame;
    MoveJ Towp31156_2_10,vmax,z30,XQ11GunTCP\WObj:=wFML2_CabFrame;
    MoveJ Towp31156_2_20,vmax,z10,XQ11GunTCP\WObj:=wFML2_CabFrame;
    SpotL wp31156_2,vmax,XQ11Gun,Sd_wp31156_2_20\QuickRelease,XQ11GunTCP\WObj:=wFML2_CabFrame;
    MoveJ Towp31206_2_10,vmax,z10,XQ11GunTCP\WObj:=wFML2_CabFrame;
    MoveJ Towp31206_2_20,vmax,z10,XQ11GunTCP\WObj:=wFML2_CabFrame;
    SpotL wp31206_2,vmax,XQ11Gun,Sd_wp31206_2_20\QuickRelease,XQ11GunTCP\WObj:=wFML2_CabFrame;
    MoveJ Towp31207_2_10,vmax,z10,XQ11GunTCP\WObj:=wFML2_CabFrame;
    MoveJ Towp31207_2_20,vmax,z10,XQ11GunTCP\WObj:=wFML2_CabFrame;
    SpotL wp31207_2,vmax,XQ11Gun,Sd_wp31207_2_20\QuickRelease,XQ11GunTCP\WObj:=wFML2_CabFrame;
    MoveJ Towp31155_2_10,vmax,z10,XQ11GunTCP\WObj:=wFML2_CabFrame;
    MoveJ Towp31155_2_20,vmax,z10,XQ11GunTCP\WObj:=wFML2_CabFrame;
    SpotL wp31155_2,vmax,XQ11Gun,Sd_wp31155_2_20\QuickRelease,XQ11GunTCP\WObj:=wFML2_CabFrame;
    MoveJ Towp31250_2_10,vmax,z10,XQ11GunTCP\WObj:=wFML2_CabFrame;
    MoveL Towp31250_2_20,vmax,z30,XQ11GunTCP\WObj:=wFML2_CabFrame;
    SpotL wp31250_2, vmax, XQ11Gun, Sd_wp31250_2_20, XQ11GunTCP\WObj:=wFML2_CabFrame;
    MoveL Towp31154_10,vmax,z30,XQ11GunTCP\WObj:=wFML2_CabFrame;
    SpotL wp31154,vmax,XQ11Gun,Sd_wp31154_20,\QuickRelease,XQ11GunTCP\WObj:=wFML2_CabFrame;
    MoveJ Towp31208_2_10,vmax,z30,XQ11GunTCP\WObj:=wFML2_CabFrame;
    MoveJ Towp31208_2_20,vmax,z30,XQ11GunTCP\WObj:=wFML2_CabFrame;
    SpotL wp31208_2,vmax,XQ11Gun,Sd_wp31208_2_20\QuickRelease,XQ11GunTCP\WObj:=wFML2_CabFrame;
    SpotL wp31249_2,vmax,XQ11Gun,Sd_wp31249_2_20\QuickRelease,XQ11GunTCP\WObj:=wFML2_CabFrame;
    SpotL wp31248_2,vmax,XQ11Gun,Sd_wp31248_2_20\QuickRelease,XQ11GunTCP\WObj:=wFML2_CabFrame;
    SpotL wp31247_2, vmax, XQ11Gun, Sd_wp31247_2_20, XQ11GunTCP\WObj:=wFML2_CabFrame;
    SpotL wp31245_2,vmax,XQ11Gun,Sd_wp31245_2_20\QuickRelease,XQ11GunTCP\WObj:=wFML2_CabFrame;
    MoveJ Towp31272_2_10,vmax,z30,XQ11GunTCP\WObj:=wFML2_CabFrame;
    MoveL Towp31272_2_20,vmax,z30,XQ11GunTCP\WObj:=wFML2_CabFrame;
    MoveJ Towp31272_2_30,vmax,z30,XQ11GunTCP\WObj:=wFML2_CabFrame;
    MoveL Towp31272_2_40,vmax,z30,XQ11GunTCP\WObj:=wFML2_CabFrame;
    SpotL wp31272_2,vmax,XQ11Gun,Sd_wp31272_2_20\QuickRelease,XQ11GunTCP\WObj:=wFML2_CabFrame;
    SpotL wp31271_2,vmax,XQ11Gun,Sd_wp31271_2_20\QuickRelease,XQ11GunTCP\WObj:=wFML2_CabFrame;
    SpotL wp31270_2,vmax,XQ11Gun,Sd_wp31270_2_20\QuickRelease,XQ11GunTCP\WObj:=wFML2_CabFrame;
    SpotL wp31269_2,vmax,XQ11Gun,Sd_wp31269_2_20\QuickRelease,XQ11GunTCP\WObj:=wFML2_CabFrame;
    SpotL wp31268_2,vmax,XQ11Gun,Sd_wp31268_2_20\QuickRelease,XQ11GunTCP\WObj:=wFML2_CabFrame;
    SpotL wp31205_2,vmax,XQ11Gun,Sd_wp31205_2_20\QuickRelease,XQ11GunTCP\WObj:=wFML2_CabFrame;
    MoveL Towp31267_2_10,vmax,z30,XQ11GunTCP\WObj:=wFML2_CabFrame;
    MoveL Towp31267_2_20,vmax,z30,XQ11GunTCP\WObj:=wFML2_CabFrame;
    SpotL wp31267_2,vmax,XQ11Gun,Sd_wp31267_2_20\QuickRelease,XQ11GunTCP\WObj:=wFML2_CabFrame;
    MoveL Frwp31267_2_10,vmax,z30,XQ11GunTCP\WObj:=wFML2_CabFrame;
    MoveL Frwp31267_2_20,vmax,z30,XQ11GunTCP\WObj:=wFML2_CabFrame;
    MoveJ Frwp31267_2_30,vmax,z30,XQ11GunTCP\WObj:=wFML2_CabFrame;
    MoveJ Frwp31267_2_40,vmax,z30,XQ11GunTCP\WObj:=wFML2_CabFrame;
    MoveJ Frwp31267_2_50,vmax,z30,XQ11GunTCP\WObj:=wFML2_CabFrame;
    MoveJ Frwp31267_2_60,vmax,z30,XQ11GunTCP\WObj:=wFML2_CabFrame;
    MoveAbsJ HomeXQ11Gun,vmax,fine,XQ11GunTCP\WObj:=wFML2_CabFrame;
ENDPROC

ENDMODULE
